// TwinCAT 3 PLC project PLC
// ProgramVersion: 3.1.4024.0
// libraries:
//   Tc2_Standard, * (Beckhoff Automation GmbH)
//   Tc2_System, * (Beckhoff Automation GmbH)
//   Tc3_Module, * (Beckhoff Automation GmbH)
// project tree:
//   Global/DUTs/ ST_GlobalStatus.TcDUT
//   Global/POUs/ MAIN.TcPOU
//   / PlcTask.TcTTO
// real-time tasks:
//   TASK PlcTask: cycle T#10ms, priority 20, ADS port 350

CONFIGURATION PLC
    RESOURCE PLC ON TwinCAT3
        TASK PlcTask(INTERVAL := T#10ms, PRIORITY := 20);
        PROGRAM MAIN WITH PlcTask : MAIN;
    END_RESOURCE
END_CONFIGURATION

// ---- Global/DUTs/ST_GlobalStatus.TcDUT
TYPE ST_GlobalStatus :
STRUCT
	nDummy							: INT;			// Some value
END_STRUCT
END_TYPE

// ---- Global/POUs/MAIN.TcPOU
PROGRAM MAIN
VAR
	stGlobalStatus				: ST_GlobalStatus;
END_VAR

stGlobalStatus.nDummy := stGlobalStatus.nDummy + 1;

END_PROGRAM
